INTERFACE I_WORD_TO_BYTES EXTENDS I_GENERAL_OBJECT

PROPERTY P_VALUE : LREAL
GET
END_GET
SET
END_SET
END_PROPERTY

PROPERTY P_X_MAX : LREAL
GET
END_GET
SET
END_SET
END_PROPERTY

PROPERTY P_X_MIN : LREAL
GET
END_GET
SET
END_SET
END_PROPERTY

PROPERTY P_Y_MAX : LREAL
GET
END_GET
SET
END_SET
END_PROPERTY

PROPERTY P_Y_MIN : LREAL
GET
END_GET
SET
END_SET
END_PROPERTY

END_INTERFACE

(* stored: Version 1.1.0.1, ProductVersion 3.1.4024.9
   Itf I_WORD_TO_BYTES: Id {a43b5e70-5fe6-4dce-a4dc-45846dc32ca6}
   Property P_VALUE: Id {bcd2043b-b63c-40d6-9ce0-b1a0aa0acd68}
   Get Get: Id {627801ee-5142-4fb4-b340-7c86e309bd09}
   Set Set: Id {dd891c25-3282-46e7-bf54-a6d32b02b039}
   Property P_X_MAX: Id {b78c3eaa-964b-4c48-92d0-37c7c0b7ffaa}
   Get Get: Id {aacf60ed-588d-4bf9-8747-5be46cc8153f}
   Set Set: Id {842ff3e2-ef13-4e71-8bb7-5d1264101f94}
   Property P_X_MIN: Id {9eccb532-fce0-44ca-b2f3-e9746fc8a442}
   Get Get: Id {14a32970-45ea-41d9-88bf-25b3663510bd}
   Set Set: Id {194d443a-5a42-40d1-9b8f-4f6d66ebb5e0}
   Property P_Y_MAX: Id {40fa60d2-c3b4-4c4d-8d6d-01cf9d60370b}
   Get Get: Id {74338adc-331a-485e-84d4-dbe12d2bbd7a}
   Set Set: Id {c8c8c7eb-c55f-4a13-bec8-ae6061489e3f}
   Property P_Y_MIN: Id {ce7075ad-edfc-4c45-b3dd-6d9b5dc86b6e}
   Get Get: Id {e004b219-9fb3-4ff5-8fc8-59bd65246952}
   Set Set: Id {280c2acb-b172-4d21-8c69-87887a94516a} *)
